FUNCTION_BLOCK Station_CAT_HMI (* Service Interface Function Block Type *)
  (* Standard: 61499-2 *)
  (* Version 0.0, 7/31/2025, Evans_A, Schneider Electric, template *)
  PACKAGE Main;
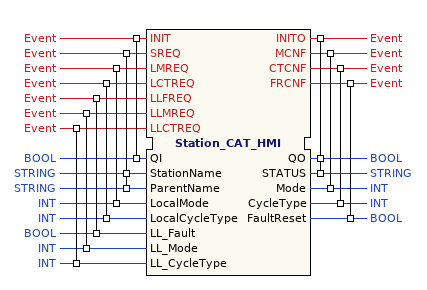
  EVENT_INPUT
    INIT WITH QI;
    SREQ WITH StationName, ParentName;
    LMREQ WITH LocalMode;
    LCTREQ WITH LocalCycleType;
    LLFREQ WITH LL_Fault;
    LLMREQ WITH LL_Mode;
    LLCTREQ WITH LL_CycleType;
  END_EVENT
  EVENT_OUTPUT
    INITO WITH QO, STATUS;
    MCNF WITH Mode;
    CTCNF WITH CycleType;
    FRCNF WITH FaultReset;
  END_EVENT
  VAR_INPUT
    QI : BOOL;
    StationName : STRING;
    ParentName : STRING;
    LocalMode : INT;
    LocalCycleType : INT;
    LL_Fault : BOOL;
    LL_Mode : INT;
    LL_CycleType : INT;
  END_VAR
  VAR_OUTPUT
    QO : BOOL; (* Event Output Qualifier *)
    STATUS : STRING; (* Service Status *)
    Mode : INT;
    CycleType : INT;
    FaultReset : BOOL;
  END_VAR
  SERVICE /
    SEQUENCE 
    END_SEQUENCE
  END_SERVICE
END_FUNCTION_BLOCK
